FUNCTION_BLOCK FB_ModuleTypeRegistry
VAR_OUTPUT
	Error : BOOL;
	ErrorMessage : STRING(255);
END_VAR
VAR
	_ModuleTypes : ARRAY[1..Param_Config.MaxModuleTypes] OF T_ModuleTypeName;
	_Adapters : ARRAY[1..Param_Config.MaxModuleTypes] OF I_ModuleConfigurationAdapter;
	_Count : UINT;
END_VAR

METHOD PUBLIC M_ClearAll : BOOL
VAR
	nAdapter : UINT;
	sAdapterError : STRING(255);
END_VAR
M_ClearAll := FALSE;
Error := FALSE;
ErrorMessage := '';
FOR nAdapter := 1 TO _Count DO
	IF NOT _Adapters[nAdapter].M_ClearAllSlots(
		ErrorMessage => sAdapterError) THEN
		Error := TRUE;
		ErrorMessage := sAdapterError;
		RETURN;
	END_IF
END_FOR
M_ClearAll := TRUE;
END_METHOD

METHOD PUBLIC M_Register : BOOL
VAR_INPUT
	ModuleTypeName : T_ModuleTypeName;
	Adapter : I_ModuleConfigurationAdapter;
END_VAR
VAR
	nIndex : UINT;
END_VAR
M_Register := FALSE;
Error := FALSE;
ErrorMessage := '';
IF (ModuleTypeName = '') OR (Adapter = 0) THEN
	Error := TRUE;
	ErrorMessage := 'A Module Type name and adapter are required.';
	RETURN;
END_IF

FOR nIndex := 1 TO _Count DO
	IF _ModuleTypes[nIndex] = ModuleTypeName THEN
		_Adapters[nIndex] := Adapter;
		M_Register := TRUE;
		RETURN;
	END_IF
END_FOR

nIndex := _Count + 1;
IF nIndex > Param_Config.MaxModuleTypes THEN
	Error := TRUE;
	ErrorMessage := 'Module type registry is full.';
	RETURN;
END_IF
_ModuleTypes[nIndex] := ModuleTypeName;
_Adapters[nIndex] := Adapter;
_Count := nIndex;
M_Register := TRUE;
END_METHOD

METHOD PUBLIC M_Resolve : I_ModuleConfigurationAdapter
VAR_INPUT
	ModuleTypeName : T_ModuleTypeName;
END_VAR
VAR
	nIndex : UINT;
END_VAR
M_Resolve := 0;
Error := FALSE;
ErrorMessage := '';
FOR nIndex := 1 TO _Count DO
	IF ModuleTypeName = _ModuleTypes[nIndex] THEN
		M_Resolve := _Adapters[nIndex];
		RETURN;
	END_IF
END_FOR
Error := TRUE;
ErrorMessage := 'Module type was not registered.';
END_METHOD

END_FUNCTION_BLOCK

(* stored: Version 1.1.0.1, ProductVersion 3.1.4026.18
   POU FB_ModuleTypeRegistry: Id {7077ad5f-0993-45c1-96b7-f6d00b53bc35}, SpecialFunc None
   Method M_ClearAll: Id {0ca10ce5-29c9-4c5f-b64c-b24780a0d046}
   Method M_Register: Id {f932ec70-80ec-4f33-8af2-c3d49daf48de}
   Method M_Resolve: Id {0e17ac2c-8fd4-42c5-a10c-27f39c8d9408} *)
